ABB RobotStudio station: Final-assignment.rspag

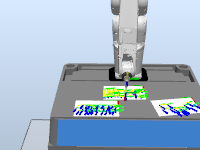
--- station ---
Station Assignment2 (saved by RobotStudio 20.4.9280.0)
Controller IRB1200_5_90, task T_ROB1: task frame (RAPID world) sits at (0, 233, 928) mm, rotated rx 0 ry 0 rz -90 deg in the station
Controller IRB1200_5_90
  mechanical unit ROB_1: IRB1200FPL_5_90_STD_02, 6 joints, base frame (0, 0, 0) mm
Layout (positions relative to the parent item):
  - IRB1200FPL_5_90_STD_02 [mechanism, from Robots\IRB1200FPL_5_90_STD_02.rslib] at (0, 233, 928) mm, rotated rx 0 ry 0 rz -90 deg; joint values [-0.0788, 0.8958, 0.2178, -0.0896, -0.8484, 0.0027] (rad or m)
  - Hardware [part]
  - Pen for irb1200 [part] at (-46.88, -430.82, 1199.31) mm, rotated rx -82.03 ry 74.58 rz 97.73 deg
Attachment: Pen for irb1200 is attached to IRB1200FPL_5_90_STD_02 / Link6

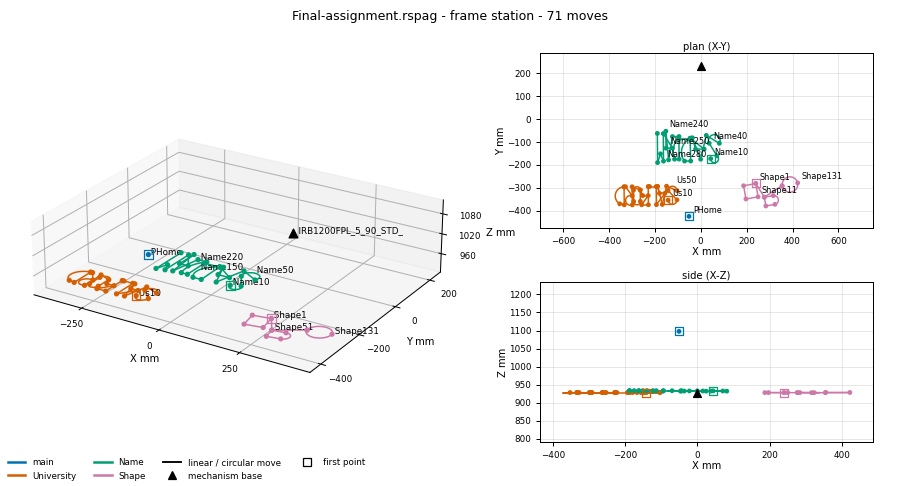
[picture p0: tool path of Final-assignment.rspag in frame station, 71 of 71 moves have a stored position in this frame; points joined in program order, loops and branches not executed]
--- Backups/IRB1200_5_90/RAPID/TASK1/PROGMOD/Module1.mod ---
MODULE Module1
	TASK PERS tooldata toolPen:=[TRUE,[[100,0,20],[1,0,0,0]],[0.1,[50,0,10],[1,0,0,0],0,0,0]];
	TASK PERS wobjdata objUniversity:=[FALSE,TRUE,"",[[459.76,-90.1561,0.0700791],[0.00418974,0.999951,0.00823316,0.00349794]],[[0,0,0],[1,0,0,0]]];
	TASK PERS wobjdata objName:=[FALSE,TRUE,"",[[234.894,103.72,2.90935],[0.00198115,0.999982,0.00391042,0.00411121]],[[0,0,0],[1,0,0,0]]];
	TASK PERS wobjdata objShape:=[FALSE,TRUE,"",[[403.819,428.003,0.0320855],[0.000825506,0.996191,0.0871904,0.00115584]],[[0,0,0],[1,0,0,0]]];
	CONST robtarget U1:=[[567.80,-371.90,0.24],[0.759116,0.0705116,0.643524,-0.0681693],[-1,-1,0,1],[9E+09,9E+09,9E+09,9E+09,9E+09,9E+09]];
	CONST robtarget Shape1:=[[75.25,204.3,0.61],[0.0797013,0.751873,-0.115924,0.644125],[0,-1,0,1],[9E+09,9E+09,9E+09,9E+09,9E+09,9E+09]];
	CONST robtarget Shape11:=[[134.52,204.3,0.61],[0.0797013,0.751873,-0.115924,0.644125],[0,-1,0,1],[9E+09,9E+09,9E+09,9E+09,9E+09,9E+09]];
	CONST robtarget Shape21:=[[134.52,258.07,0.61],[0.0797013,0.751873,-0.115924,0.644124],[0,-1,0,1],[9E+09,9E+09,9E+09,9E+09,9E+09,9E+09]];
	CONST robtarget Shape31:=[[76.07,258.07,0.61],[0.0797013,0.751873,-0.115924,0.644124],[0,-1,0,1],[9E+09,9E+09,9E+09,9E+09,9E+09,9E+09]];
	CONST robtarget Shape41:=[[76.07,203.99,0.61],[0.0797013,0.751873,-0.115924,0.644124],[0,-1,0,1],[9E+09,9E+09,9E+09,9E+09,9E+09,9E+09]];
	CONST robtarget Shape51:=[[140.55,177.88,0.61],[0.0797013,0.751873,-0.115924,0.644124],[0,-1,0,1],[9E+09,9E+09,9E+09,9E+09,9E+09,9E+09]];
	CONST robtarget Shape61:=[[179.51,177.88,0.61],[0.0797013,0.751873,-0.115924,0.644124],[0,-1,0,1],[9E+09,9E+09,9E+09,9E+09,9E+09,9E+09]];
	CONST robtarget Shape71:=[[179.51,137.89,0.61],[0.0797013,0.751874,-0.115924,0.644124],[0,0,0,1],[9E+09,9E+09,9E+09,9E+09,9E+09,9E+09]];
	CONST robtarget Shape91:=[[140.74,138.08,0.62],[0.0797018,0.75187,-0.115923,0.644128],[0,0,0,1],[9E+09,9E+09,9E+09,9E+09,9E+09,9E+09]];
	CONST robtarget Shape81:=[[159.85,119.43,0.61],[0.0797008,0.751874,-0.115924,0.644123],[0,0,0,1],[9E+09,9E+09,9E+09,9E+09,9E+09,9E+09]];
	CONST robtarget Shape101:=[[140.74,177.91,0.62],[0.0797018,0.751869,-0.115923,0.644129],[0,-1,0,1],[9E+09,9E+09,9E+09,9E+09,9E+09,9E+09]];
	CONST robtarget Shape111:=[[104.54,93.24,0.62],[0.0797017,0.751869,-0.115923,0.644129],[0,0,0,1],[9E+09,9E+09,9E+09,9E+09,9E+09,9E+09]];
	CONST robtarget Shape131:=[[104.76,24.12,-0.18],[0.0797004,0.751873,-0.115924,0.644125],[0,0,-1,1],[9E+09,9E+09,9E+09,9E+09,9E+09,9E+09]];
	CONST robtarget Shape121:=[[139.17,58.59,0.61],[0.0797008,0.751873,-0.115924,0.644124],[0,0,-1,1],[9E+09,9E+09,9E+09,9E+09,9E+09,9E+09]];
	CONST robtarget Shape151:=[[107.28,92.33,-0.38],[0.0797034,0.751867,-0.115923,0.644132],[0,0,0,1],[9E+09,9E+09,9E+09,9E+09,9E+09,9E+09]];
	CONST robtarget Shape141:=[[72.42,58.87,-0.38],[0.0797025,0.751867,-0.115922,0.644131],[0,0,0,1],[9E+09,9E+09,9E+09,9E+09,9E+09,9E+09]];
	CONST robtarget PHome:=[[656.76,-50.64,169.64],[0.606705,-0.0115484,0.794713,-0.0143731],[-1,-1,0,1],[9E+09,9E+09,9E+09,9E+09,9E+09,9E+09]];
	CONST robtarget Us10:=[[586.44,-141.41,0.2],[0.761056,0.0207771,0.641038,-0.0971184],[-1,-1,-1,1],[9E+09,9E+09,9E+09,9E+09,9E+09,9E+09]];
	CONST robtarget Us20:=[[604.42,-121.6,0.2],[0.761056,0.0207772,0.641039,-0.0971184],[-1,-1,-1,1],[9E+09,9E+09,9E+09,9E+09,9E+09,9E+09]];
	CONST robtarget Us30:=[[584.82,-103.02,0.27],[0.781259,0.0638459,0.617543,-0.064799],[-1,0,0,1],[9E+09,9E+09,9E+09,9E+09,9E+09,9E+09]];
	CONST robtarget Us40:=[[544.61,-141.98,0.27],[0.78126,0.0638457,0.617541,-0.0647992],[-1,-1,0,1],[9E+09,9E+09,9E+09,9E+09,9E+09,9E+09]];
	CONST robtarget Us50:=[[525.71,-123.01,0.27],[0.781259,0.0638459,0.617543,-0.0647991],[-1,-1,0,1],[9E+09,9E+09,9E+09,9E+09,9E+09,9E+09]];
	CONST robtarget Us60:=[[544.79,-103.36,0.27],[0.78126,0.0638458,0.617542,-0.0647992],[-1,-1,0,1],[9E+09,9E+09,9E+09,9E+09,9E+09,9E+09]];
	CONST robtarget Names10:=[[169.06,61.25,0.08],[0.0538504,0.619983,-0.0626806,0.780252],[0,-1,0,1],[9E+09,9E+09,9E+09,9E+09,9E+09,9E+09]];
	CONST robtarget Names20:=[[187.05,38.51,0.08],[0.0538504,0.619982,-0.0626807,0.780252],[0,-1,0,1],[9E+09,9E+09,9E+09,9E+09,9E+09,9E+09]];
	CONST robtarget Names30:=[[153.74,34.70,0.08],[0.0538504,0.619983,-0.0626807,0.780252],[0,-1,0,1],[9E+09,9E+09,9E+09,9E+09,9E+09,9E+09]];
	CONST robtarget Names40:=[[102.36,67.48,-0.25],[0.0538501,0.619984,-0.0626807,0.780251],[0,-1,-1,1],[9E+09,9E+09,9E+09,9E+09,9E+09,9E+09]];
	CONST robtarget Names50:=[[74.08,53.58,-0.25],[0.0538502,0.619984,-0.0626808,0.78025],[0,-1,0,1],[9E+09,9E+09,9E+09,9E+09,9E+09,9E+09]];
	CONST robtarget Names60:=[[102.02,22.46,-0.25],[0.0538504,0.619984,-0.0626808,0.78025],[0,0,0,1],[9E+09,9E+09,9E+09,9E+09,9E+09,9E+09]];
	CONST robtarget Name10:=[[170.04,61.2,-0.25],[0.0538501,0.619984,-0.0626806,0.780251],[0,-1,0,1],[9E+09,9E+09,9E+09,9E+09,9E+09,9E+09]];
	CONST robtarget Name30:=[[157.69,34.25,-0.25],[0.05385,0.619984,-0.0626808,0.780251],[0,-1,0,1],[9E+09,9E+09,9E+09,9E+09,9E+09,9E+09]];
	CONST robtarget Name20:=[[187.31,38.48,-0.25],[0.0538501,0.619983,-0.0626808,0.780252],[0,-1,0,1],[9E+09,9E+09,9E+09,9E+09,9E+09,9E+09]];
	CONST robtarget Name40:=[[102.94,67.27,-0.25],[0.05385,0.619987,-0.0626809,0.780249],[0,-1,-1,1],[9E+09,9E+09,9E+09,9E+09,9E+09,9E+09]];
	CONST robtarget Name60:=[[103.65,22.99,-0.25],[0.0538502,0.619985,-0.0626808,0.78025],[0,0,0,1],[9E+09,9E+09,9E+09,9E+09,9E+09,9E+09]];
	CONST robtarget Name50:=[[66.07,49.64,-0.25],[0.05385,0.619986,-0.062681,0.780249],[0,-1,0,1],[9E+09,9E+09,9E+09,9E+09,9E+09,9E+09]];
	CONST robtarget Name70:=[[68.83,79.77,-0.25],[0.0538502,0.619985,-0.0626807,0.78025],[0,-1,-1,1],[9E+09,9E+09,9E+09,9E+09,9E+09,9E+09]];
	CONST robtarget Name80:=[[172.22,105.02,-0.25],[0.0538499,0.619983,-0.0626809,0.780251],[-1,-1,-1,1],[9E+09,9E+09,9E+09,9E+09,9E+09,9E+09]];
	CONST robtarget Name90:=[[78.53,140.59,-0.25],[0.0538496,0.619983,-0.062681,0.780251],[-1,-1,-1,1],[9E+09,9E+09,9E+09,9E+09,9E+09,9E+09]];
	CONST robtarget Name100:=[[128.11,126.59,-0.25],[0.0538498,0.619983,-0.0626812,0.780251],[-1,-1,-1,1],[9E+09,9E+09,9E+09,9E+09,9E+09,9E+09]];
	CONST robtarget Name110:=[[128.11,89.49,-0.25],[0.0538498,0.619983,-0.0626812,0.780252],[-1,-1,-1,1],[9E+09,9E+09,9E+09,9E+09,9E+09,9E+09]];
	CONST robtarget Name120:=[[80.1,150.53,-0.25],[0.0538495,0.619982,-0.0626814,0.780252],[-1,-1,-1,1],[9E+09,9E+09,9E+09,9E+09,9E+09,9E+09]];
	CONST robtarget Name130:=[[179.87,148.38,-0.25],[0.0538495,0.619982,-0.0626815,0.780252],[-1,-1,-1,1],[9E+09,9E+09,9E+09,9E+09,9E+09,9E+09]];
	CONST robtarget Name140:=[[179.87,175.03,-0.25],[0.0538495,0.619982,-0.0626815,0.780252],[-1,-1,-1,1],[9E+09,9E+09,9E+09,9E+09,9E+09,9E+09]];
	CONST robtarget Name160:=[[83.29,150.4,-0.25],[0.0538502,0.619982,-0.062681,0.780252],[-1,-1,-1,1],[9E+09,9E+09,9E+09,9E+09,9E+09,9E+09]];
	CONST robtarget Name150:=[[132.64,187.79,-0.25],[0.0538496,0.619982,-0.0626813,0.780252],[-1,-1,-1,1],[9E+09,9E+09,9E+09,9E+09,9E+09,9E+09]];
	CONST robtarget Name170:=[[83.29,198.88,-0.25],[0.0538503,0.619982,-0.0626808,0.780252],[-1,-1,-1,1],[9E+09,9E+09,9E+09,9E+09,9E+09,9E+09]];
	CONST robtarget Name180:=[[171.29,198.88,-0.25],[0.0538503,0.619983,-0.0626808,0.780252],[-1,-1,-1,1],[9E+09,9E+09,9E+09,9E+09,9E+09,9E+09]];
	CONST robtarget Name190:=[[171.29,218.61,-0.25],[0.0538503,0.619983,-0.0626808,0.780252],[-1,-1,-1,1],[9E+09,9E+09,9E+09,9E+09,9E+09,9E+09]];
	CONST robtarget Name210:=[[72.7,198.46,-0.32],[0.0538505,0.619983,-0.0626802,0.780251],[-1,-1,-1,1],[9E+09,9E+09,9E+09,9E+09,9E+09,9E+09]];
	CONST robtarget Name200:=[[135.69,223.94,-0.25],[0.0538499,0.619983,-0.0626806,0.780252],[-1,-1,-1,1],[9E+09,9E+09,9E+09,9E+09,9E+09,9E+09]];
	CONST robtarget Name220:=[[72.7,227.21,-0.32],[0.0538505,0.619984,-0.0626801,0.780251],[-1,-1,-1,1],[9E+09,9E+09,9E+09,9E+09,9E+09,9E+09]];
	CONST robtarget Name230:=[[174.16,244.75,-0.32],[0.0538505,0.619984,-0.0626802,0.780251],[-1,-1,-1,1],[9E+09,9E+09,9E+09,9E+09,9E+09,9E+09]];
	CONST robtarget Name240:=[[48.98,255.47,-0.32],[0.05385,0.619983,-0.0626803,0.780251],[-1,-1,-1,1],[9E+09,9E+09,9E+09,9E+09,9E+09,9E+09]];
	CONST robtarget Name250:=[[123.11,255.47,-0.32],[0.0538499,0.619983,-0.0626804,0.780251],[-1,-1,-1,1],[9E+09,9E+09,9E+09,9E+09,9E+09,9E+09]];
	CONST robtarget Name260:=[[123.11,227.49,-0.32],[0.0538497,0.619983,-0.0626805,0.780251],[-1,-1,-1,1],[9E+09,9E+09,9E+09,9E+09,9E+09,9E+09]];
	CONST robtarget Name270:=[[59.41,266.83,-0.32],[0.0538496,0.619983,-0.0626805,0.780251],[-1,-1,-1,1],[9E+09,9E+09,9E+09,9E+09,9E+09,9E+09]];
	CONST robtarget Name280:=[[179.39,266.83,-0.32],[0.0538496,0.619983,-0.0626805,0.780251],[-1,-1,-1,1],[9E+09,9E+09,9E+09,9E+09,9E+09,9E+09]];
	CONST robtarget Name290:=[[147.31,279.78,-0.32],[0.0538496,0.619983,-0.0626805,0.780251],[-1,-1,-1,1],[9E+09,9E+09,9E+09,9E+09,9E+09,9E+09]];
	CONST robtarget Name300:=[[185.43,292.67,-0.32],[0.0538498,0.619983,-0.0626803,0.780251],[-1,-1,-1,1],[9E+09,9E+09,9E+09,9E+09,9E+09,9E+09]];
	CONST robtarget Name310:=[[58.43,292.67,-0.32],[0.0538497,0.619983,-0.0626802,0.780251],[-1,-1,-1,1],[9E+09,9E+09,9E+09,9E+09,9E+09,9E+09]];
	VAR num MyChoice:=0;
	VAR num NumUni:=0;
	VAR num NumShape:=0;
	VAR num NumName:=0;
    !***********************************************************
    !
    ! Module:  Module1
    !
    ! Description:
    !   <Insert description here>
    !
    ! Author: saddamcoder
    !
    ! Version: 1.0
    !
    !***********************************************************


    !***********************************************************
    !
    ! Procedure main
    !
    !   This is the entry point of your program
    !
    !***********************************************************
    PROC main()
        !Add your code here
        MoveJ PHome, v100, z50, toolPen;
        TPErase;
        TPWrite "Drawing Demo work";
        TPWrite "Number of university name="\Num:=NumUni;
        TPWrite "Number of shape="\Num:=NumShape;
        TPWrite "Number of Name="\Num:=NumName;
        TPReadFK MyChoice, "Which want to draw", "University Name", "Shapes", "My Name", stEmpty, stEmpty;
        TEST Mychoice
        CASE 1:
        	University;
        CASE 2:
        	Shape;
        CASE 3:
        	Name;
        ENDTEST
    ENDPROC
	PROC University()
		MoveL Us10, v100, z50, toolPen;
		MoveC Us20, Us30, v100, fine, toolPen;
		MoveL Us40, v100, fine, toolPen;
		MoveC Us50, Us60, v100, fine, toolPen;
		MoveL [[525.59,-148.44,0.08],[0.759116,0.0705105,0.643524,-0.068173],[-1,-1,0,1],[9E+09,9E+09,9E+09,9E+09,9E+09,9E+09]], v100, z50, toolPen;
		MoveL [[604.83,-167.01,0.08],[0.759121,0.0705099,0.643519,-0.0681739],[-1,-1,0,1],[9E+09,9E+09,9E+09,9E+09,9E+09,9E+09]], v100, z50, toolPen;
		MoveL [[526.16,-187.2,0.08],[0.759122,0.0705097,0.643517,-0.0681741],[-1,-1,0,1],[9E+09,9E+09,9E+09,9E+09,9E+09,9E+09]],v100,z50,toolPen;
		MoveL [[556.75,-179.33,0.25],[0.759121,0.0705099,0.643518,-0.068174],[-1,-1,0,1],[9E+09,9E+09,9E+09,9E+09,9E+09,9E+09]], v100, z50, toolPen;
		MoveL [[556.75,-155.74,0.25],[0.759121,0.0705099,0.643519,-0.0681739],[-1,-1,0,1],[9E+09,9E+09,9E+09,9E+09,9E+09,9E+09]], v100, z50, toolPen;
		MoveL [[605.68,-192.57,0.25],[0.759122,0.0705096,0.643517,-0.0681742],[-1,-1,0,1],[9E+09,9E+09,9E+09,9E+09,9E+09,9E+09]], v100, fine, toolPen;
		MoveL [[526.95,-193.33,0.25],[0.759122,0.0705096,0.643517,-0.0681742],[-1,-1,0,1],[9E+09,9E+09,9E+09,9E+09,9E+09,9E+09]], v100, z50, toolPen;
		MoveL [[526.95,-222.68,0.25],[0.759122,0.0705095,0.643517,-0.0681743],[-1,-1,0,1],[9E+09,9E+09,9E+09,9E+09,9E+09,9E+09]], v100, z50, toolPen;
		MoveL [[526.95,-228.34,0.25],[0.759123,0.0705095,0.643517,-0.0681744],[-1,-1,0,1],[9E+09,9E+09,9E+09,9E+09,9E+09,9E+09]], v100, z50, toolPen;
		MoveL [[606.19,-227.53,0.25],[0.759122,0.0705095,0.643517,-0.0681744],[-1,-1,0,1],[9E+09,9E+09,9E+09,9E+09,9E+09,9E+09]], v100, z50, toolPen;
		MoveL [[606.19,-256.81,0.25],[0.759123,0.0705095,0.643517,-0.0681744],[-1,-1,0,1],[9E+09,9E+09,9E+09,9E+09,9E+09,9E+09]], v100, fine, toolPen;
		MoveL [[566.24,-228.14,0.25],[0.759122,0.0705095,0.643517,-0.0681744],[-1,-1,0,1],[9E+09,9E+09,9E+09,9E+09,9E+09,9E+09]], v100, fine, toolPen;
		MoveL [[566.24,-252.21,0.25],[0.759123,0.0705094,0.643516,-0.0681744],[-1,-1,0,1],[9E+09,9E+09,9E+09,9E+09,9E+09,9E+09]], v100, z50, toolPen;
		MoveL [[541.86,-263.05,0.25],[0.759124,0.0705092,0.643515,-0.0681747],[-1,-1,0,1],[9E+09,9E+09,9E+09,9E+09,9E+09,9E+09]], v100, z50, toolPen;
		MoveL [[591.58,-262.53,0.25],[0.759124,0.0705093,0.643515,-0.0681747],[-1,-1,0,1],[9E+09,9E+09,9E+09,9E+09,9E+09,9E+09]], v100, z50, toolPen;
		MoveC [[606.54,-276.92,0.25],[0.759126,0.0705084,0.643512,-0.0681753],[-1,-1,0,1],[9E+09,9E+09,9E+09,9E+09,9E+09,9E+09]],[[592,-291.62,0.25],[0.759127,0.070508,0.643511,-0.0681753],[-1,-1,0,1],[9E+09,9E+09,9E+09,9E+09,9E+09,9E+09]],v100,z10,toolPen;
		MoveL [[542.49,-292.25,0.25],[0.759127,0.0705079,0.643511,-0.0681751],[-1,-1,0,1],[9E+09,9E+09,9E+09,9E+09,9E+09,9E+09]], v100, z50, toolPen;
		MoveC [[527.57,-278.08,0.25],[0.759124,0.0705092,0.643515,-0.0681743],[-1,-1,0,1],[9E+09,9E+09,9E+09,9E+09,9E+09,9E+09]], [[542.03,-263.15,0.25],[0.759123,0.0705098,0.643515,-0.0681748],[-1,-1,0,1],[9E+09,9E+09,9E+09,9E+09,9E+09,9E+09]], v100, z10, toolPen;
		MoveL [[527.94,-298.44,0.25],[0.759124,0.0705097,0.643515,-0.0681749],[-1,-1,0,1],[9E+09,9E+09,9E+09,9E+09,9E+09,9E+09]], v100, fine, toolPen;
		MoveL [[606.88,-297.52,0.25],[0.759124,0.0705096,0.643515,-0.0681753],[-1,-1,0,1],[9E+09,9E+09,9E+09,9E+09,9E+09,9E+09]], v100, z50, toolPen;
		MoveC [[587.64,-326.67,0.25],[0.759125,0.0705092,0.643514,-0.0681751],[-1,-1,0,1],[9E+09,9E+09,9E+09,9E+09,9E+09,9E+09]], [[567.38,-297.98,0.25],[0.759122,0.0705104,0.643517,-0.0681743],[-1,-1,0,1],[9E+09,9E+09,9E+09,9E+09,9E+09,9E+09]], v100, fine, toolPen;
		MoveL [[527.81,-327.13,0.25],[0.759122,0.0705096,0.643517,-0.0681729],[-1,-1,0,1],[9E+09,9E+09,9E+09,9E+09,9E+09,9E+09]], v100, fine, toolPen;
		MoveL [[528.73,-333.39,0.25],[0.759123,0.0705093,0.643517,-0.0681731],[-1,-1,0,1],[9E+09,9E+09,9E+09,9E+09,9E+09,9E+09]], v100, z50, toolPen;
		MoveL [[606.52,-332.55,0.24],[0.759116,0.0705123,0.643525,-0.06817],[-1,-1,0,1],[9E+09,9E+09,9E+09,9E+09,9E+09,9E+09]], v100, z50, toolPen;
		MoveL [[602.16,-352.31,0.24],[0.759116,0.070512,0.643524,-0.06817],[-1,-1,0,1],[9E+09,9E+09,9E+09,9E+09,9E+09,9E+09]], v100, z50, toolPen;
		MoveC [[567.8,-371.9,0.24],[0.759116,0.0705116,0.643524,-0.0681693],[-1,-1,0,1],[9E+09,9E+09,9E+09,9E+09,9E+09,9E+09]],[[528.16,-333.29,0.24],[0.759115,0.0705127,0.643526,-0.0681699],[-1,-1,0,1],[9E+09,9E+09,9E+09,9E+09,9E+09,9E+09]],v100,z10,toolPen;
		Incr NumUni;
	ENDPROC
	PROC Name()
        !Add your code here
        MoveL Name10, v100, fine, toolPen\WObj:=objName;
        MoveC Name20, Name30, v100, fine, toolPen\WObj:=objName;
        MoveL Name40, v100, fine, toolPen\WObj:=objName;
        MoveC Name50, Name60, v100, fine, toolPen\WObj:=objName;
        MoveL Name70, v100, fine, toolPen\WObj:=objName;
        MoveL Name80, v100, fine, toolPen\WObj:=objName;
        MoveL Name90, v100, fine, toolPen\WObj:=objName;
        MoveL Name100, v100, fine, toolPen\WObj:=objName;
        MoveL Name110, v100, fine, toolPen\WObj:=objName;
        MoveL Name120, v100, fine, toolPen\WObj:=objName;
        MoveL Name130, v100, fine, toolPen\WObj:=objName;
        MoveL Name140, v100, fine, toolPen\WObj:=objName;
        MoveC Name150, Name160, v100, fine, toolPen\WObj:=objName;
        MoveL Name170, v100, fine, toolPen\WObj:=objName;
        MoveL Name180, v100, fine, toolPen\WObj:=objName;
        MoveL Name190, v100, fine, toolPen\WObj:=objName;
        MoveC Name200, Name210, v100, fine, toolPen\WObj:=objName;
        MoveL Name220, v100, fine, toolPen\WObj:=objName;
        MoveL Name230, v100, fine, toolPen\WObj:=objName;
        MoveL Name240, v100, fine, toolPen\WObj:=objName;
        MoveL Name250, v100, z50, toolPen\WObj:=objName;
        MoveL Name260, v100, z50, toolPen\WObj:=objName;
        MoveL Name270, v100, z50, toolPen\WObj:=objName;
        MoveL Name280, v100, z50, toolPen\WObj:=objName;
        MoveL Name290, v100, z50, toolPen\WObj:=objName;
        MoveL Name300, v100, z50, toolPen\WObj:=objName;
        MoveL Name310, v100, z50, toolPen\WObj:=objName;
        Incr NumName;
	ENDPROC
	PROC Shape()
		MoveL Shape1, v100, z50, toolPen\WObj:=objShape;
		MoveL Shape11, v100, fine, toolPen\WObj:=objShape;
		MoveL Shape21, v100, fine, toolPen\WObj:=objShape;
		MoveL Shape31, v100, fine, toolPen\WObj:=objShape;
		MoveL Shape41, v100, fine, toolPen\WObj:=objShape;
		WaitTime 2;
		MoveL Shape51, v100, z50, toolPen\WObj:=objShape;
		MoveL Shape61, v100, z50, toolPen\WObj:=objShape;
		MoveL Shape71, v100, z50, toolPen\WObj:=objShape;
		MoveC Shape81, Shape91, v100, z10, toolPen\WObj:=objShape;
		MoveL Shape101, v100, z50, toolPen\WObj:=objShape;
		WaitTime 2;
		MoveL Shape111, v100, z50, toolPen\WObj:=objShape;
		MoveC Shape121, Shape131, v100, z10, toolPen\WObj:=objShape;
		MoveC Shape141, Shape151, v100, z10, toolPen\WObj:=objShape;
		Incr NumShape;
	ENDPROC
ENDMODULE

--- Backups/IRB1200_5_90/RAPID/TASK1/SYSMOD/LINKEDM.sys ---
%%%
  VERSION:1
  LANGUAGE:ENGLISH
%%%

MODULE LINKEDM (SYSMODULE)

! FOLLOWER
!     Name of electronically linked follower axis used by operator at teach pendent.
      PERS string l_f_axis_name{5}       :=  ["",  "", "", "", ""];

!     Name of the mechanical unit for follower axis.
      PERS string l_f_mecunt_n{5}  :=  ["", "", "", "", ""];

!     Linked follower axis number in the mechanical unit (first axis in mech. unit is number 1).
      PERS num l_f_axis_no{5}      :=  [0,          0,   0,  0,  0];

! MASTER
!     Name of the mechanical unit for linked master axis.
      PERS string l_m_mecunt_n{5} :=  ["", "", "", "", ""];

!     Linked master axis number in the mechanical unit (first axis in mech. unit is number 1).
!     See axis number table in documentation for different master mechanical units.
      PERS num l_m_axis_no{5}     :=  [0,  0,  0,  0,  0];

! POSITION OFFSET
!     The increase of the allowed offset position between the master and follower
!     positions, used when starting AUTO mode. As soon as the offset is decreased
!     the old configurated parameter is used.
!     Example: 3 => the configurated value of allowed offset is increased 3 times.
      PERS num offset_ratio{5}       :=  [10,  10,   10,  10,  10];

! SPEED RATIO
!     Speed_ratio used in AUTO and JOG modes [ very_slow   slow    normal    fast]
!     Value 1 = max allowed manual speed.
      CONST num speed_ratio {20}      := [0.01, 0.01, 0.01, 0.01, 0.01,
                                          0.05, 0.05, 0.05, 0.05, 0.05,
                                          0.20, 0.20, 0.20, 0.20, 0.20,
                                          1.00, 1.00, 1.00, 1.00, 1.00];

! STEP SIZE
!     Displacement position used in JOG mode for each activation of positive or
!     negative movement.                  [very_short    short   normal   long]
!     Unit degees or meter.
      CONST num displacement {20}     := [0.001, 0.001, 0.001, 0.001, 0.001,
                                          0.005, 0.005, 0.005, 0.005, 0.005,
                                          0.020, 0.020, 0.020, 0.020, 0.020,
                                          0.100, 0.100, 0.100, 0.100, 0.100];


!-------------------------------------------------------------
 PROC Linked_m ()
      Linked_m_exe ;
 ENDPROC
ENDMODULE
